(* PLC project IEC_61131-1, IEC_61131-1 1.0 *)
(* stored: creationDateTime 2008-12-14T16:21:19, contentDescription Load data from Source: name_file: file 1 field name_file_CSV: file many field, productRelease 1.0, modificationDateTime 2020-10-08T10:21:58, version 0.2 *)

TYPE StateMachine : (STANDBY, START, STOP);
END_TYPE

TYPE datatype0 : STRUCT
  _1NJ20T001 : STRING := '_1NJ20T001.csv';
  _1CV20T001 : STRING := '_1CV20T001.csv';
  Rashod_1 : STRING := 'Rashod_1.csv';
  Rashod_2 : STRING := 'Rashod_2.csv';
  PID_1 : STRING := 'PID_1.csv';
  PID_2 : STRING := 'PID_2.csv';
  PID_3 : STRING := 'PID_3.csv';
  IN : STRING := 'IN';
  OUT : STRING := 'OUT';
  IBM : STRING := 'IBM.csv';
  Amper : STRING := 'Amper';
  Amper_A : STRING := 'Amper_A';
  Amper_B : STRING := 'Amper_B';
  Amper_C : STRING := 'Amper_C';
END_STRUCT;
END_TYPE

FUNCTION get_val_row : STRING
  VAR_INPUT
    nameFile : STRING;
    nameField : STRING;
  END_VAR

            get_val_row:=CONCAT('get_val_row("',nameFile,'","',nameField,'")');
          
END_FUNCTION

FUNCTION_BLOCK get_value_CSV
  VAR
    pyTrigger : BOOL;
  END_VAR
  VAR_INPUT
    nameFile : STRING;
    nameField : STRING := 'IN';
  END_VAR
  VAR_OUTPUT
    value_outFB : REAL;  (* Value out *)
  END_VAR
  VAR
    python_eval0 : python_eval;
  END_VAR
  VAR  (* added by the conversion: wires and edge detectors of the diagram *)
    _NOT2_OUT : BOOL;
  END_VAR

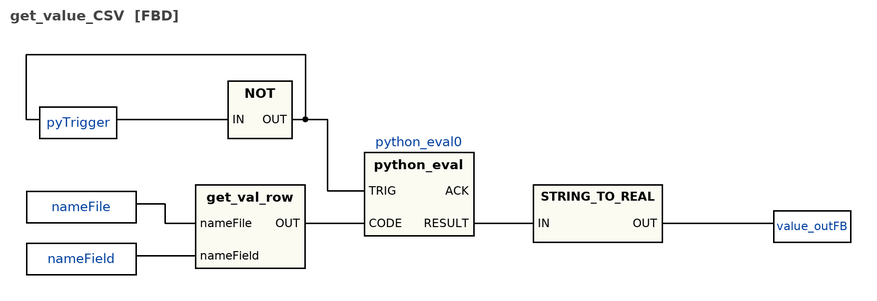
(* FBD diagram, written out as Structured Text *)
_NOT2_OUT := NOT pyTrigger;
pyTrigger := _NOT2_OUT;
python_eval0(TRIG := _NOT2_OUT, CODE := get_val_row(nameFile, nameField));
value_outFB := STRING_TO_REAL(python_eval0.RESULT);
END_FUNCTION_BLOCK

FUNCTION set_val_row : STRING
  VAR_INPUT
    nameFile : STRING;
    nameField : STRING;
    value : REAL;
  END_VAR
  VAR
    str_temp : STRING;
  END_VAR

            set_val_row:=CONCAT('set_val_row("',CONCAT(nameFile,'","',nameField),'","',REAL_TO_STRING(value),'")');

          
END_FUNCTION

FUNCTION_BLOCK set_value_CSV
  VAR
    pyTrigger : BOOL;
  END_VAR
  VAR_INPUT
    nameFile : STRING;
    nameField : STRING := 'IN';
  END_VAR
  VAR_OUTPUT
    i_status : INT;  (* Value out *)
  END_VAR
  VAR
    python_eval0 : python_eval;
  END_VAR
  VAR_INPUT
    value_IN : REAL;
  END_VAR
  VAR  (* added by the conversion: wires and edge detectors of the diagram *)
    _NOT2_OUT : BOOL;
  END_VAR

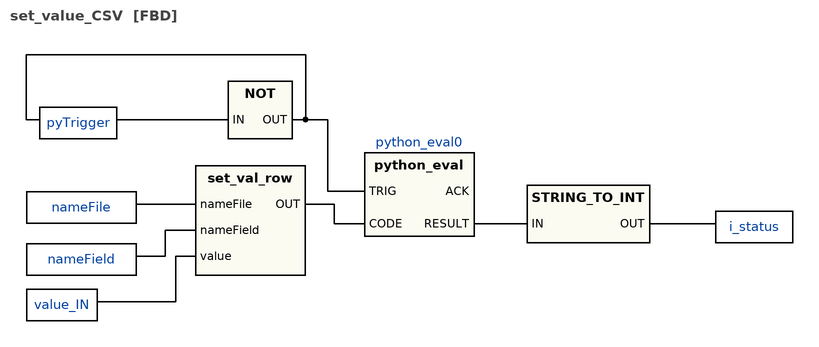
(* FBD diagram, written out as Structured Text *)
_NOT2_OUT := NOT pyTrigger;
pyTrigger := _NOT2_OUT;
python_eval0(TRIG := _NOT2_OUT, CODE := set_val_row(nameFile, nameField, value_IN));
i_status := STRING_TO_INT(python_eval0.RESULT);
END_FUNCTION_BLOCK

FUNCTION openCSV : STRING
  VAR_INPUT
    arg : STRING;
  END_VAR

            openCSV:=CONCAT('openCSV("',arg,'")');

          
END_FUNCTION

FUNCTION readSignalCSV : STRING
  VAR_INPUT
    nameFile : STRING;
    i_status : STRING;
  END_VAR

            readSignalCSV:=CONCAT('readSignalCSV("',i_status,'","',nameFile,'")');
          
END_FUNCTION

FUNCTION writeSignalCSV : STRING
  VAR_INPUT
    nameFile : STRING;
  END_VAR

            writeSignalCSV:=CONCAT('writeCSV("',nameFile,'")');
          
END_FUNCTION

FUNCTION_BLOCK SourceFromFileCSV
  VAR
    pyTrigger : BOOL := TRUE;
    pyTriggerOpenCSV : BOOL := TRUE;
  END_VAR
  VAR_INPUT
    nameFileFB : STRING := 'unknow.csv';
  END_VAR
  VAR_OUTPUT
    i_status_readSignal_CSV : INT;  (* Value out *)
    i_status_writeSignal_CSV : INT;  (* Status write CSV *)
  END_VAR
  VAR
    python_eval0 : python_eval;
    str_func : STRING;
    python_eval1 : python_eval;
    python_eval2 : python_eval;
    con_writeCSV : STRING;
  END_VAR
  VAR  (* added by the conversion: wires and edge detectors of the diagram *)
    _NOT2_OUT : BOOL;
  END_VAR

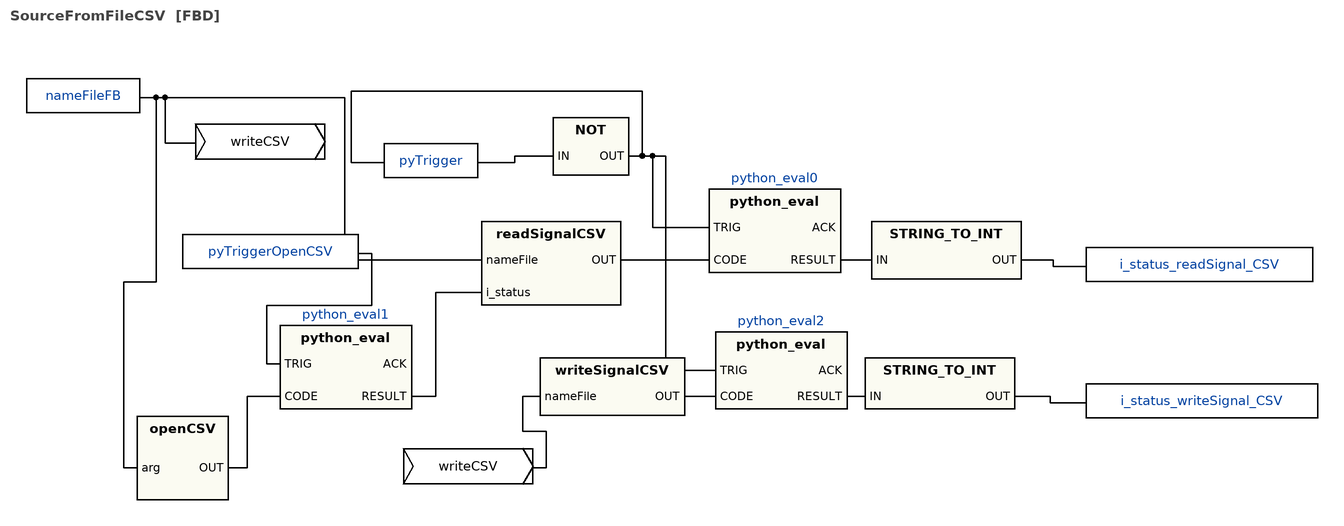
(* FBD diagram, written out as Structured Text *)
_NOT2_OUT := NOT pyTrigger;
pyTrigger := _NOT2_OUT;
python_eval1(TRIG := pyTriggerOpenCSV, CODE := openCSV(nameFileFB));
python_eval0(TRIG := _NOT2_OUT, CODE := readSignalCSV(nameFileFB, python_eval1.RESULT));
i_status_readSignal_CSV := STRING_TO_INT(python_eval0.RESULT);
python_eval2(TRIG := _NOT2_OUT, CODE := writeSignalCSV(nameFileFB));
i_status_writeSignal_CSV := STRING_TO_INT(python_eval2.RESULT);
END_FUNCTION_BLOCK

(* Testing fron CSV-files *)
PROGRAM TestCSV_v_3
  VAR
    pyTriger : BOOL := FALSE;
    Tags : datatype0;
    result : STRING := 'Initial String';
    i_status_read_CSV : INT := 0;
    i_status_read_CSV1 : INT := 0;
    i_status_write_CSV : INT := 0;
    i_status_open_CSV : INT := 0;
    val_out_1 : REAL := 0.0;
    val_out_2 : REAL := 0.0;
    val_out_3 : REAL := 0.0;
    val_IN : datatype0;
    SourceFromFileCSV0 : SourceFromFileCSV;
    get_value_CSV0 : get_value_CSV;
    get_value_CSV1 : get_value_CSV;
    set_value_CSV0 : set_value_CSV;
    set_value_CSV1 : set_value_CSV;
    set_value_CSV2 : set_value_CSV;
    INTEGRAL0 : INTEGRAL;
    run : BOOL := true;
    cycle : STRING := '0:0:1';
    triger : BOOL := false;
  END_VAR
  VAR  (* added by the conversion: wires and edge detectors of the diagram *)
    _NOT22_OUT : BOOL;
  END_VAR

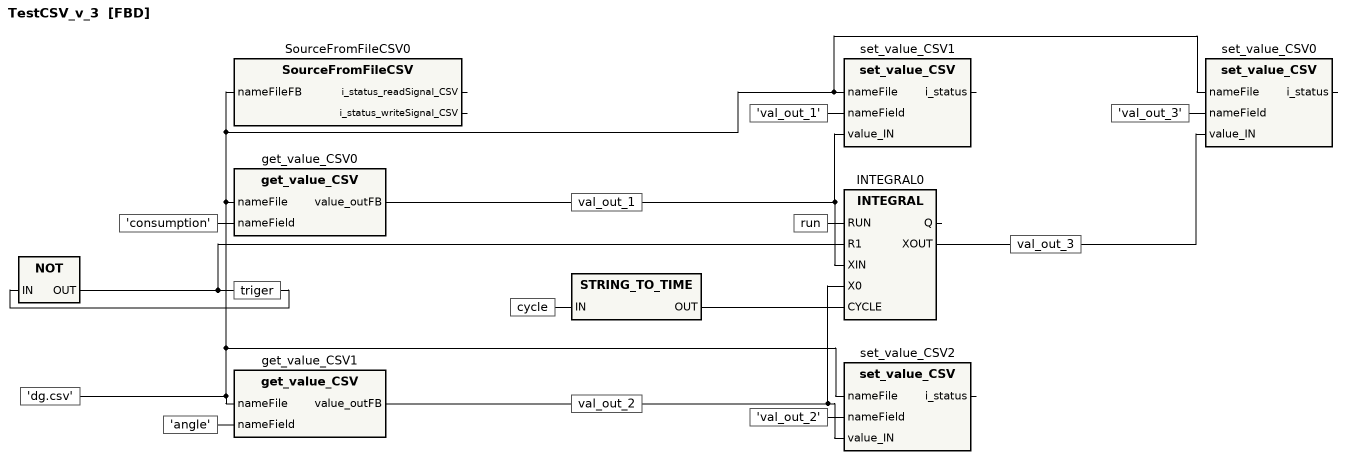
(* FBD diagram, written out as Structured Text *)
get_value_CSV0(nameFile := 'dg.csv', nameField := 'consumption');
val_out_1 := get_value_CSV0.value_outFB;
_NOT22_OUT := NOT triger;
INTEGRAL0(RUN := run, R1 := _NOT22_OUT, XIN := val_out_1, X0 := val_out_2, CYCLE := STRING_TO_TIME(cycle));
val_out_3 := INTEGRAL0.XOUT;
get_value_CSV1(nameFile := 'dg.csv', nameField := 'angle');
val_out_2 := get_value_CSV1.value_outFB;
triger := _NOT22_OUT;
SourceFromFileCSV0(nameFileFB := 'dg.csv');
set_value_CSV0(nameFile := 'dg.csv', nameField := 'val_out_3', value_IN := val_out_3);
set_value_CSV1(nameFile := 'dg.csv', nameField := 'val_out_1', value_IN := val_out_1);
set_value_CSV2(nameFile := 'dg.csv', nameField := 'val_out_2', value_IN := val_out_2);
END_PROGRAM

(* Testing fron CSV-files *)
PROGRAM TestCSV_v_2
  VAR
    pyTriger : BOOL := FALSE;
    Tags : datatype0;
    result : STRING := 'Initial String';
    i_status_read_CSV : INT := 0;
    i_status_read_CSV1 : INT := 0;
    i_status_write_CSV : INT := 0;
    i_status_open_CSV : INT := 0;
    val_out_1 : REAL := 0.0;
    val_out_2 : REAL := 0.0;
    val_out_3 : REAL := 0.0;
    val_out_4 : REAL := 0.0;
    val_out_5 : REAL := 0.0;
    val_out_6 : REAL := 0.0;
    val_out_7 : REAL := 0.0;
    val_out_8 : REAL := 0.0;
    val_out_9 : REAL := 0.0;
    val_out_10 : REAL := 0.0;
    val_out_11 : REAL := 10.0;
    val_IN : datatype0;
    SourceFromFileCSV0 : SourceFromFileCSV;
    get_value_CSV0 : get_value_CSV;
    get_value_CSV1 : get_value_CSV;
    set_value_CSV0 : set_value_CSV;
    set_value_CSV1 : set_value_CSV;
    set_value_CSV2 : set_value_CSV;
  END_VAR

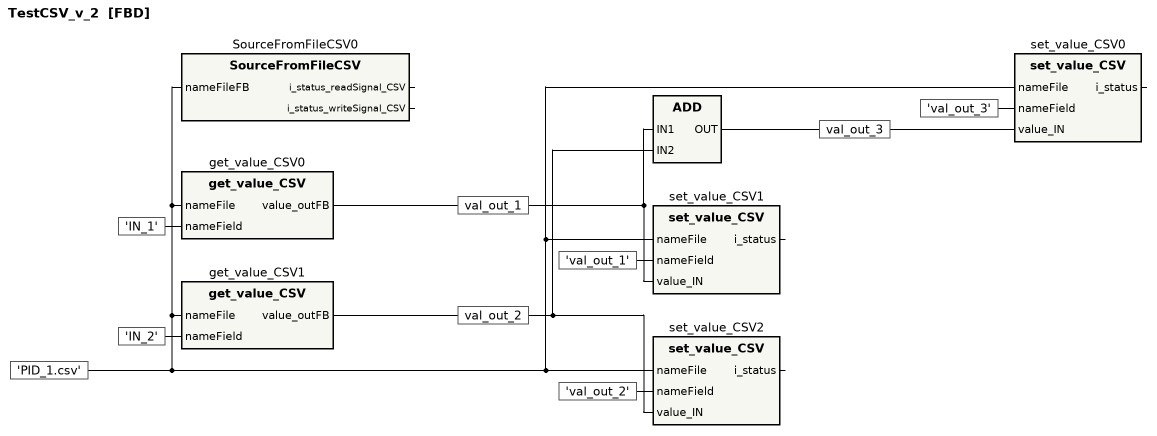
(* FBD diagram, written out as Structured Text *)
get_value_CSV0(nameFile := 'PID_1.csv', nameField := 'IN_1');
val_out_1 := get_value_CSV0.value_outFB;
val_out_3 := val_out_1 + val_out_2;
get_value_CSV1(nameFile := 'PID_1.csv', nameField := 'IN_2');
val_out_2 := get_value_CSV1.value_outFB;
SourceFromFileCSV0(nameFileFB := 'PID_1.csv');
set_value_CSV0(nameFile := 'PID_1.csv', nameField := 'val_out_3', value_IN := val_out_3);
set_value_CSV1(nameFile := 'PID_1.csv', nameField := 'val_out_1', value_IN := val_out_1);
set_value_CSV2(nameFile := 'PID_1.csv', nameField := 'val_out_2', value_IN := val_out_2);
END_PROGRAM

(* Testing fron CSV-files *)
PROGRAM TestCSV_v_1
  VAR
    pyTriger : BOOL := FALSE;
    Tags : datatype0;
    result : STRING;
    i_status_read_CSV : INT;
    i_status_read_CSV1 : INT;
    i_status_write_CSV : INT;
    i_status_open_CSV : INT;
    val_out_1 : REAL;
    val_out_2 : REAL;
    val_out_3 : REAL;
    val_out_4 : REAL;
    val_out_5 : REAL;
    val_out_6 : REAL;
    val_out_7 : REAL;
    val_out_8 : REAL;
    val_out_9 : REAL;
    val_out_10 : REAL;
    val_IN : datatype0;
    get_value_CSV0 : get_value_CSV;
    get_value_CSV1 : get_value_CSV;
    SourceFromFileCSV0 : SourceFromFileCSV;
    SourceFromFileCSV1 : SourceFromFileCSV;
    get_value_CSV2 : get_value_CSV;
    get_value_CSV3 : get_value_CSV;
    set_value_CSV0 : set_value_CSV;
    set_value_CSV1 : set_value_CSV;
    set_value_CSV2 : set_value_CSV;
    set_value_CSV3 : set_value_CSV;
    set_value_CSV4 : set_value_CSV;
    set_value_CSV5 : set_value_CSV;
  END_VAR

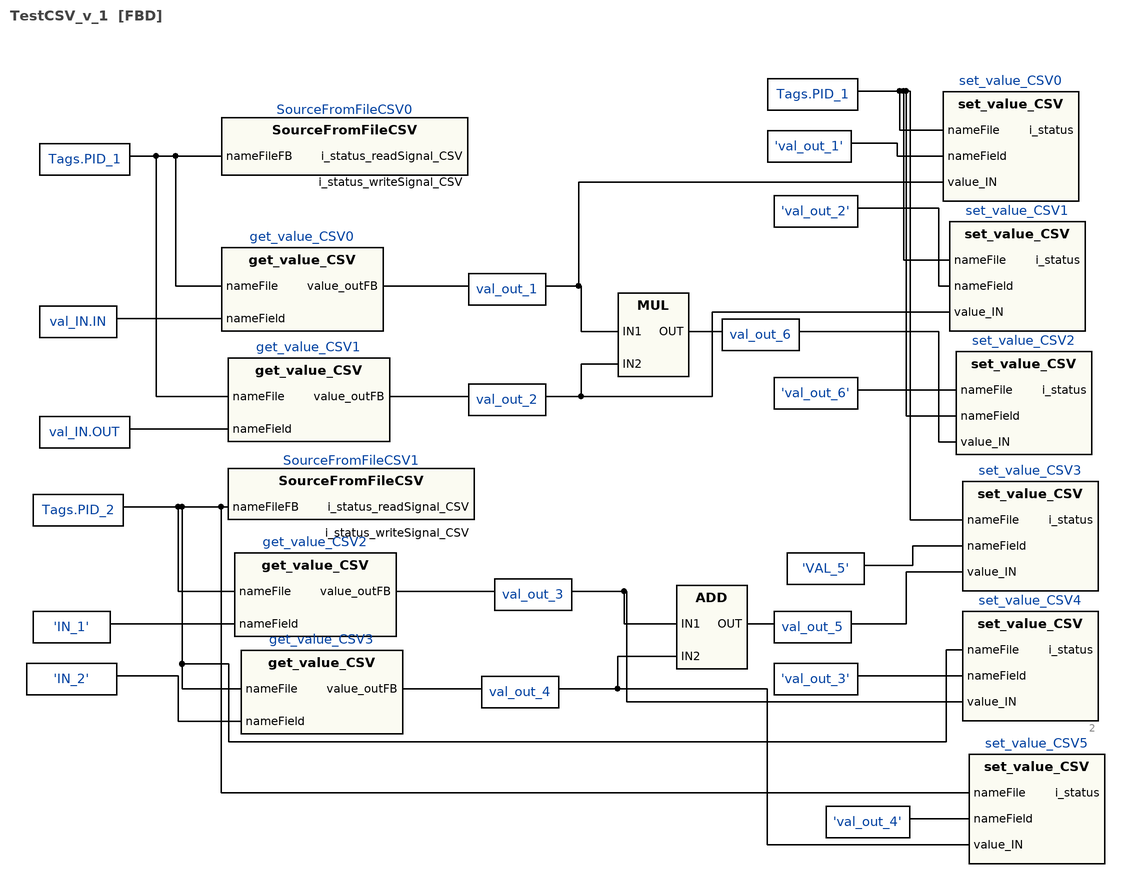
(* FBD diagram, written out as Structured Text *)
set_value_CSV4(nameFile := Tags.PID_2, nameField := 'val_out_3', value_IN := val_out_3);
get_value_CSV0(nameFile := Tags.PID_1, nameField := val_IN.IN);
val_out_1 := get_value_CSV0.value_outFB;
val_out_6 := val_out_1 * val_out_2;
get_value_CSV1(nameFile := Tags.PID_1, nameField := val_IN.OUT);
val_out_2 := get_value_CSV1.value_outFB;
get_value_CSV2(nameFile := Tags.PID_2, nameField := 'IN_1');
val_out_3 := get_value_CSV2.value_outFB;
val_out_5 := val_out_3 + val_out_4;
get_value_CSV3(nameFile := Tags.PID_2, nameField := 'IN_2');
val_out_4 := get_value_CSV3.value_outFB;
set_value_CSV0(nameFile := Tags.PID_1, nameField := 'val_out_1', value_IN := val_out_1);
SourceFromFileCSV0(nameFileFB := Tags.PID_1);
set_value_CSV1(nameFile := Tags.PID_1, nameField := 'val_out_2', value_IN := val_out_2);
set_value_CSV2(nameFile := Tags.PID_1, nameField := 'val_out_6', value_IN := val_out_6);
SourceFromFileCSV1(nameFileFB := Tags.PID_2);
set_value_CSV3(nameFile := Tags.PID_1, nameField := 'VAL_5', value_IN := val_out_5);
set_value_CSV5(nameFile := Tags.PID_2, nameField := 'val_out_4', value_IN := val_out_4);
END_PROGRAM

FUNCTION readSignal : STRING
  VAR_INPUT
    arg : STRING;
  END_VAR

            readSignal:=CONCAT('readSignal("',arg,'")');

          
END_FUNCTION

FUNCTION_BLOCK SourceFromFile
  VAR
    pyTrigger : BOOL;
  END_VAR
  VAR_INPUT
    nameFileFB : STRING := '_1NJ20T001.csv';
  END_VAR
  VAR_OUTPUT
    value_outFB : REAL;  (* Value out *)
  END_VAR
  VAR
    python_eval0 : python_eval;
    str_func : STRING;
  END_VAR
  VAR  (* added by the conversion: wires and edge detectors of the diagram *)
    _NOT2_OUT : BOOL;
  END_VAR

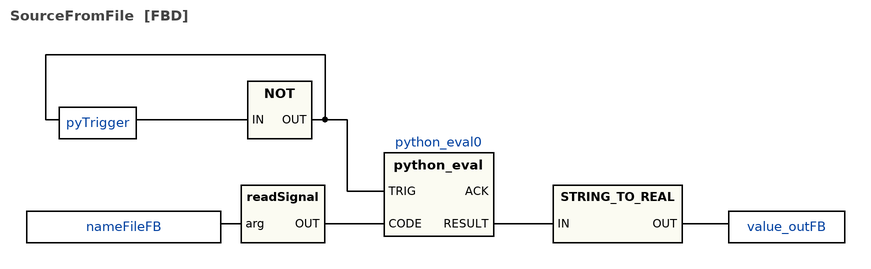
(* FBD diagram, written out as Structured Text *)
_NOT2_OUT := NOT pyTrigger;
pyTrigger := _NOT2_OUT;
python_eval0(TRIG := _NOT2_OUT, CODE := readSignal(nameFileFB));
value_outFB := STRING_TO_REAL(python_eval0.RESULT);
END_FUNCTION_BLOCK

PROGRAM TestSourceFromFile
  VAR_INPUT
    NameFile : STRING := '_1NJ20T002.csv';
  END_VAR
  VAR
    NameFileDataType : datatype0;
  END_VAR
  VAR_EXTERNAL
    ValueOUT : REAL;
  END_VAR
  VAR_OUTPUT
    value_1 : REAL;
  END_VAR
  VAR
    SourceFromFile0 : SourceFromFile;
    SourceFromFile1 : SourceFromFile;
    SourceFromFile2 : SourceFromFile;
  END_VAR

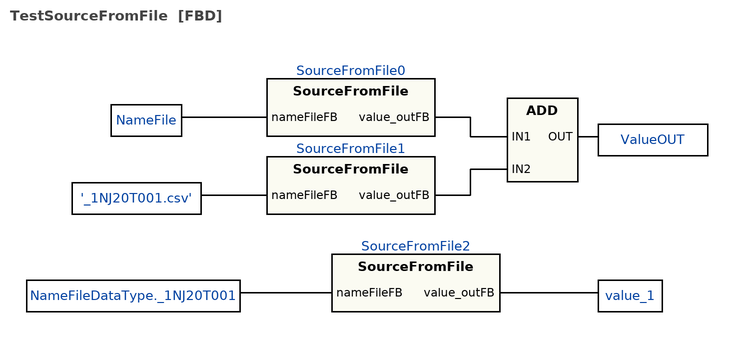
(* FBD diagram, written out as Structured Text *)
SourceFromFile0(nameFileFB := NameFile);
SourceFromFile1(nameFileFB := '_1NJ20T001.csv');
ValueOUT := SourceFromFile0.value_outFB + SourceFromFile1.value_outFB;
SourceFromFile2(nameFileFB := NameFileDataType._1NJ20T001);
value_1 := SourceFromFile2.value_outFB;
END_PROGRAM

PROGRAM DG
  VAR
    SourceFromFile0 : SourceFromFile;
    SourceFromFile1 : SourceFromFile;
    IN1 : datatype0;
    IN2 : datatype0;
    Exp_IN : INT := 3;
    Val_OUT : REAL;
    Rashod_1_IN : REAL;
    Rashod_2_IN : REAL;
  END_VAR

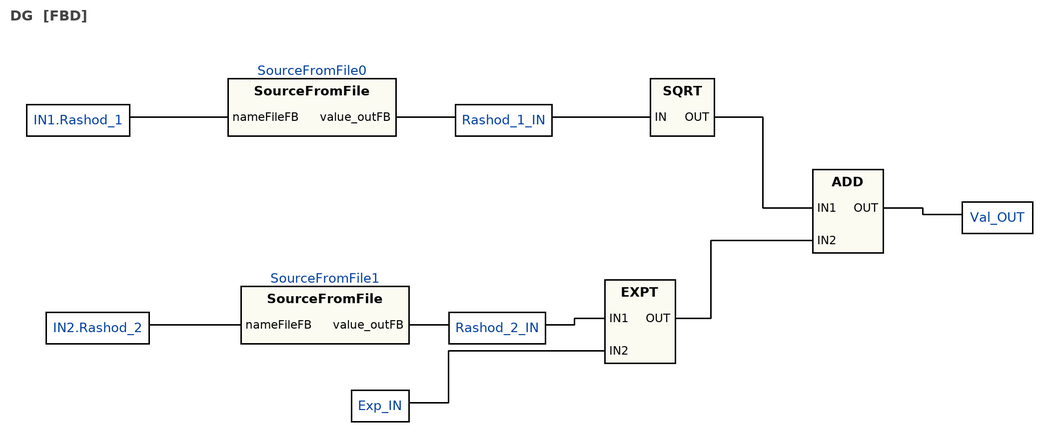
(* FBD diagram, written out as Structured Text *)
SourceFromFile0(nameFileFB := IN1.Rashod_1);
Rashod_1_IN := SourceFromFile0.value_outFB;
Val_OUT := SQRT(Rashod_1_IN) + EXPT(Rashod_2_IN, Exp_IN);
SourceFromFile1(nameFileFB := IN2.Rashod_2);
Rashod_2_IN := SourceFromFile1.value_outFB;
END_PROGRAM

(* Testing fron CSV-files *)
PROGRAM TestCSV
  VAR
    pyTriger : BOOL := FALSE;
    Tags : datatype0;
    result : STRING;
    i_status_read_CSV : INT;
    i_status_read_CSV1 : INT;
    i_status_write_CSV : INT;
    i_status_open_CSV : INT;
    val_out_1 : REAL;
    val_out_2 : REAL;
    val_out_3 : REAL;
    val_out_4 : REAL;
    val_out_5 : REAL;
    val_out_6 : REAL;
    val_out_7 : REAL;
    val_out_8 : REAL;
    val_out_9 : REAL;
    val_out_10 : REAL;
    val_out_12 : REAL;
    val_IN : datatype0;
    get_value_CSV0 : get_value_CSV;
    get_value_CSV1 : get_value_CSV;
    SourceFromFileCSV0 : SourceFromFileCSV;
    SourceFromFileCSV1 : SourceFromFileCSV;
    get_value_CSV2 : get_value_CSV;
    get_value_CSV3 : get_value_CSV;
    set_value_CSV0 : set_value_CSV;
    set_value_CSV1 : set_value_CSV;
    set_value_CSV2 : set_value_CSV;
    set_value_CSV3 : set_value_CSV;
  END_VAR

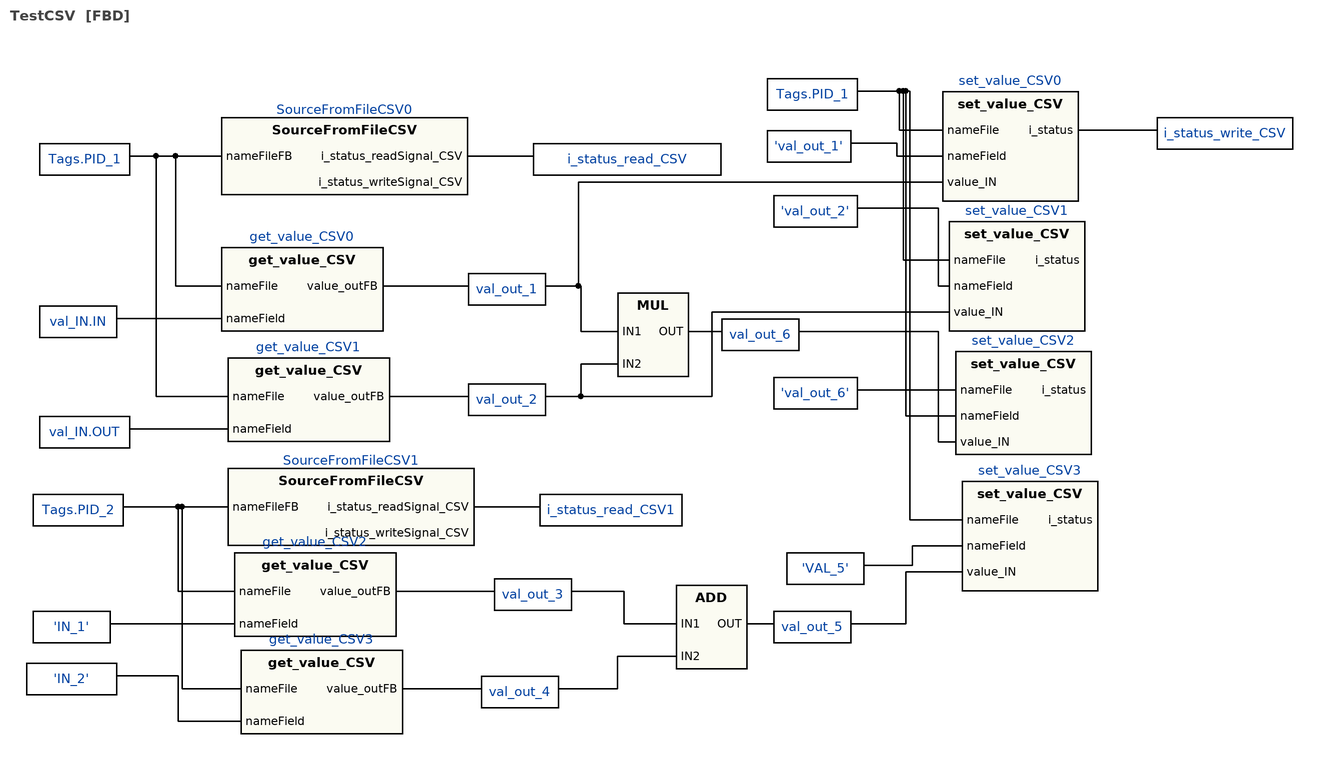
(* FBD diagram, written out as Structured Text *)
set_value_CSV0(nameFile := Tags.PID_1, nameField := 'val_out_1', value_IN := val_out_1);
i_status_write_CSV := set_value_CSV0.i_status;
SourceFromFileCSV0(nameFileFB := Tags.PID_1);
i_status_read_CSV := SourceFromFileCSV0.i_status_readSignal_CSV;
get_value_CSV0(nameFile := Tags.PID_1, nameField := val_IN.IN);
val_out_1 := get_value_CSV0.value_outFB;
val_out_6 := val_out_1 * val_out_2;
get_value_CSV1(nameFile := Tags.PID_1, nameField := val_IN.OUT);
val_out_2 := get_value_CSV1.value_outFB;
SourceFromFileCSV1(nameFileFB := Tags.PID_2);
i_status_read_CSV1 := SourceFromFileCSV1.i_status_readSignal_CSV;
get_value_CSV2(nameFile := Tags.PID_2, nameField := 'IN_1');
val_out_3 := get_value_CSV2.value_outFB;
val_out_5 := val_out_3 + val_out_4;
get_value_CSV3(nameFile := Tags.PID_2, nameField := 'IN_2');
val_out_4 := get_value_CSV3.value_outFB;
set_value_CSV1(nameFile := Tags.PID_1, nameField := 'val_out_2', value_IN := val_out_2);
set_value_CSV2(nameFile := Tags.PID_1, nameField := 'val_out_6', value_IN := val_out_6);
set_value_CSV3(nameFile := Tags.PID_1, nameField := 'VAL_5', value_IN := val_out_5);
END_PROGRAM

CONFIGURATION config
  VAR_GLOBAL
    Global_RS : RS;
  END_VAR
  RESOURCE res_pytest ON PLC
    VAR_GLOBAL
      ValueOUT : REAL;
    END_VAR
    TASK pytest_task(INTERVAL := T#1s0ms, PRIORITY := 0);
    PROGRAM MyProg : TestCSV_v_3;
  END_RESOURCE
END_CONFIGURATION
